Staubli VAL3: refreshStatic.pgx

program refreshStatic()
  local string l_sMenu
  local num i
  local string l_sInstruction
  local num l_nSize
  local string l_sMessage
  local mdesc l_mDesc
  local num l_nTcpAction
  local string l_sName
  local string l_sEmpty
  local bool l_bStop
  local num l_nEmpty
  local num l_nIndexTool
  local string l_sType
  local string l_sData
begin
 // cls()
  title("编辑-1号石墨舟A面取片-第1槽/6槽")
  l_sMenu="权限,,,,,吸片,放片,保存"
  // define the menu
  call use:stringToArray(l_sMenu,sMenu)
  sMenu[0]=sMenu+sTitle
  call use:setMenu(sMenu,true,2)

////  call use:listadd(sList)



//  //
//  l_sMenu="1,2,,,,,,"
//  call use:stringToArray(l_sMenu,sMenu)
//  call use:setMenu(sMenu,false,3)
//  call use:getMenu(sMenu,bButton)

//  call use:setSizeList(0,0,38,12)
//  call use:listcreate("第1槽/8槽")
//  //
//  call use:listadd(sList)
//  //
//  // refresh the list
//  call use:selectNewField(nSelected,nIndex,nView)
//  //

//    title("111")
//    l_sMenu="模拟,复位,,,,,,"
//  // define the menu
//  call use:stringToArray(l_sMenu,sMenu)
//    // set the menu
//  call use:setMenu(sMenu,true,2)
//  call use:getMenu(sMenu,bButton)
end
